FUNCTION_BLOCK FB_CylinderTempDiag EXTENDS FB_CylinderTemp
VAR_INPUT
	fTempMin			:		LREAL;					// Global value:	minimal allowed cylinder temperature for temperature monitoring
	fTempMax			:		LREAL;					// Global value:	maximal allowed cylinder temperature for temperature monitoring
END_VAR
VAR_OUTPUT
	bError				:		BOOL;					// Error signal		(diagnosed from temperature monitoring)
	sErrorMsg			:		STRING;					// Error message
	nErrorID			:		UDINT;					// Error ID
END_VAR
VAR
END_VAR

METHOD Diag
VAR_INPUT
END_VAR
IF fTempCurrent > fTempMax OR fTempCurrent < fTempMin	THEN
	bError	:=	TRUE;
ELSE
	bError	:=	FALSE;
END_IF

IF bError	THEN
	IF		fTempCurrent > fTempMax	THEN
			sErrorMsg	:=		'Temperature above maximum';
			nErrorID	:=		94;
	ELSIF	fTempCurrent < fTempMin	THEN
			sErrorMsg	:=		'Temperature below minimum';
			nErrorID	:=		93;
	END_IF
ELSE
	sErrorMsg		:=	'';
	nErrorID		:=	0;
END_IF
END_METHOD

METHOD Reset
VAR_INPUT
END_VAR
SUPER^.Reset();

bError			:=		FALSE;
sErrorMsg		:=		'';
nErrorID		:=		0;
END_METHOD

METHOD PROTECTED StateMachine
VAR_INPUT
	bBasePosReq		:	BOOL;
	bWorkPosReq		:	BOOL;
END_VAR
IF NOT bError THEN
	// Calling StateMachine() method of parental class FB_Cylinder
	SUPER^.StateMachine(	bBasePosReq			:=		bBasePosReq,
							bWorkPosReq			:=		bWorkPosReq);
	
	// Diagnosis evaluation by every movement of cylinder							
	Diag();
END_IF
END_METHOD

END_FUNCTION_BLOCK

(* stored: Version 1.1.0.1, ProductVersion 3.1.4024.15
   POU FB_CylinderTempDiag: Id {e448bdd6-215b-4669-ac4e-f2fc2daf26a0}, SpecialFunc None
   Method Diag: Id {073f25e6-e23c-42a2-91dd-fe77e9b46a98}
   Method Reset: Id {e1d57925-d9dd-485b-a81e-091364fdb114}
   Method StateMachine: Id {10be3644-55f4-4439-8c92-9ae5d4b3e963} *)
